// TIA Portal V19 export
VAR_GLOBAL   // PLC tag table "Default tag table"
   RHSystemClockByte AT %IB0 : Byte;   // Recieved from RH System as heartbeat
   InputByte1 AT %IB1 : Byte;
   InputByte2 AT %IB2 : Byte;
   InputByte3 AT %IB3 : Byte;
   InputByte4 AT %IB4 : Byte;
   InputByte5 AT %IB5 : Byte;
   InputByte6 AT %IB6 : Byte;
   InputByte7 AT %IB7 : Byte;
   InputByte8 AT %IB8 : Byte;
   InputByte9 AT %IB9 : Byte;
   InputByte10 AT %IB10 : Byte;
   LocalSystemClockbyte AT %QB0 : Byte;   // Sent to RH System as heartbeat
   OutputByte1 AT %QB1 : Byte;
   OutputByte2 AT %QB2 : Byte;
   OutputByte3 AT %QB3 : Byte;
   OutputByte4 AT %QB4 : Byte;
   OutputByte5 AT %QB5 : Byte;
   OutputByte6 AT %QB6 : Byte;
   OutputByte7 AT %QB7 : Byte;
   OutputByte8 AT %QB8 : Byte;
   OutputByte9 AT %QB9 : Byte;
   OutputByte10 AT %QB10 : Byte;
   System_Byte AT %MB1 : Byte;
   FirstScan AT %M1.0 : Bool;
   DiagStatusUpdate AT %M1.1 : Bool;
   AlwaysTRUE AT %M1.2 : Bool;
   AlwaysFALSE AT %M1.3 : Bool;
   Clock_Byte AT %MB0 : Byte;
   Clock_10Hz AT %M0.0 : Bool;
   Clock_5Hz AT %M0.1 : Bool;
   "Clock_2.5Hz" AT %M0.2 : Bool;
   Clock_2Hz AT %M0.3 : Bool;
   "Clock_1.25Hz" AT %M0.4 : Bool;
   Clock_1Hz AT %M0.5 : Bool;
   "Clock_0.625Hz" AT %M0.6 : Bool;
   "Clock_0.5Hz" AT %M0.7 : Bool;
   GreenPushButton AT %IB27 : Byte;
   BluePushButton AT %IB34 : Byte;
   SelectorSwitch AT %IB35 : Byte;
   RedPushButton AT %IB36 : Byte;
   GreenPushButtonLamp AT %QB32 : Byte;
   BluePushButtonLamp AT %QB33 : Byte;
   SelectorSwitchLamp AT %QB34 : Byte;
   RedPushButtonLamp AT %QB35 : Byte;
   "EstopF-In_ModuleByte1" AT %IB28 : Byte;
   "EstopF-In_ModuleByte2" AT %IB29 : Byte;
   "EstopF-In_ModuleByte3" AT %IB30 : Byte;
   "EstopF-In_ModuleByte4" AT %IB31 : Byte;
   "EstopF-In_ModuleByte5" AT %IB32 : Byte;
   "EstopF-In_ModuleByte6" AT %IB33 : Byte;
   "Estop-FOut_ModuleByte1" AT %QB28 : Byte;
   "Estop-FOut_ModuleByte2" AT %QB29 : Byte;
   "Estop-FOut_ModuleByte3" AT %QB30 : Byte;
   "Estop-FOut_ModuleByte4" AT %QB31 : Byte;
END_VAR
